// TIA Portal V20 export
TYPE "LER_typeMobileRFIDConfrolNode"
// stored: Access Published
   STRUCT
      commands { ExternalAccessible := 'False'; ExternalVisible := 'False'; ExternalWritable := 'False'} : "LER_typeMobileRFIDCommands";
      monitoring { ExternalAccessible := 'False'; ExternalVisible := 'False'; ExternalWritable := 'False'} : "LER_typeMobileRFIDMonitoring";
   END_STRUCT;
END_TYPE
